// Mitsubishi GX Works2 project: Sequence   PLC: Q03UDV

PROGRAM MAIN
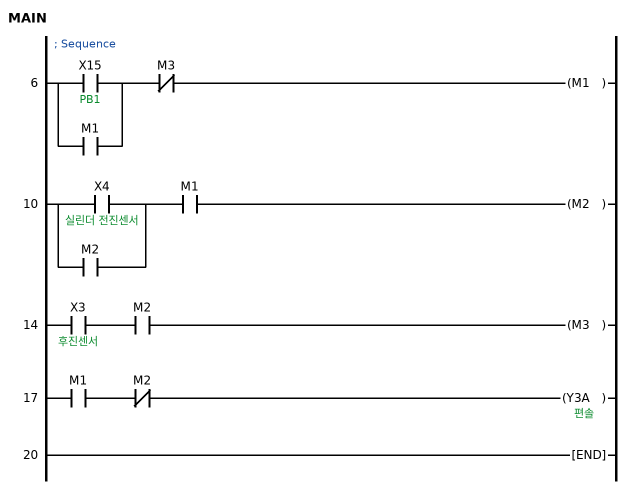
; Sequence
6     LD      X15  ; PB1
      OR      M1
      ANI     M3
      OUT     M1
10    LD      X4  ; 실린더 전진센서
      OR      M2
      AND     M1
      OUT     M2
14    LD      X3  ; 후진센서
      AND     M2
      OUT     M3
17    LD      M1
      ANI     M2
      OUT     Y3A  ; 편솔
20    END
END_PROGRAM
